// TIA Portal V20 export
TYPE "LER_typeJobInterface"
// stored: Access Published
   STRUCT
      Request { ExternalWritable := 'False'} : Array[0..99] of Bool;
      Ready { ExternalWritable := 'False'} : Array[0..99] of Bool;
      Busy : Array[0..99] of Bool;
      Done { ExternalWritable := 'False'} : Array[0..99] of Bool;
      workingDone { ExternalWritable := 'False'} : Array[0..99] of Bool;
   END_STRUCT;
END_TYPE
